(* Logix 5000 project; controller R5_CSS vendor 1 type 14 code 74 rev 19.11; software revision 19.01; part 20 of 20 *)
(* tags used below, declared in another part *)
   FC101 : FLOW_CONTROL;   // QUENCH BASIN FLOW TRANSMITTER CONTROL
   FC101_PIDE : PID_ENHANCED;
   FC140 : FLOW_CONTROL;
   FC140A : FLOW_CONTROL;   // QUENCH TOWER UPPER SPRAY FLOW CONTROL
   FC140B : FLOW_CONTROL;   // QUENCH TOWER LOWER SPRAY FLOW CONTROL
   FC365 : FLOW_CONTROL;   // COALESCER PROCESS IMPURITY FLOW CONTROL
   FT140_TOTAL_FLOW : REAL;
   InputMax_IF8 : REAL;
   InputMin_IF8 : REAL;
   LC101 : LEVEL_CONTROL;   // QUENCH TOWER BASIN LIT
   MyTime : DINT[10];
   P303A : PUMP_CONTROL;
   P303B : PUMP_CONTROL;
   PC132 : PRESSURE_CONTROL;
   PC132_PID : PID;
   PID_FCV365 : PID;
   PID_TCV108_Flow : PID;
   RandomNumber : REAL;
   RandomNumberDint : DINT;
   TC108 : TEMP_CONTROL;   // QUENCH TOWER EXIT GAS TEMPERATURE CONTROL
   TIMER : TIMER[50];   // HX A TIMER FOR START

PROGRAM Simulate   (* main routine MainProgram *)
VAR
   BasinFlowBalance : REAL := 94.5125;
   BasinFlowBalanceAdd : REAL := 0.45176974;
   BasinFlowBalanceAddSCLP : SCLP := (Input := 0.45176974, InputMax := 38.0, ScaledMax := 16000.0, Output := 190.21884);
   BasinFlowBalanceRawAdd : REAL := 190.21884;
   BasinFlowBalanceTmr : TIMER := (PRE := 1000);
   FC140_PID_Sim : AI_Simulate := (ControlVariable := 20.0, AI_Counts := 4025, RandomNumber := 0.637, PID_P := 1.0, PID_I := 1.0, ScaledMin := 4000, ScaledMax := 20000, PID_CV_Min := 20.0, PID_CV_Max := 100.0, UpdateSec := 1.0, DirectActing := 1);
   FC140_SUM : DINT := 4037;
   FC140_SUM_Flow : REAL := 0.46250153;
   FC140_SUM_sclp : SCLP := (Input := 4000.0, InputMin := 4000.0, InputMax := 20000.0, ScaledMax := 200.0);
   FC140A_Flow : REAL := 0.18500061;
   FC140A_SUM : SCLP := (Input := 0.125, InputMax := 200.0, ScaledMin := 4000.0, ScaledMax := 20000.0, Output := 4010.0);
   FC140B_Flow : REAL := 0.27750093;
   FC140B_SUM : SCLP := (Input := 0.25499955, InputMax := 200.0, ScaledMin := 4000.0, ScaledMax := 20000.0, Output := 4020.4);
   FC365_FT_SIM_ENABLE : BOOL;
   FC365_PID_Sim : AI_Simulate := (ControlVariable := 50.0, AI_Counts := 12033, RandomNumber := 0.149, PID_P := 1.0, PID_I := 1.0, ScaledMin := 4000, ScaledMax := 20000, PID_CV_Max := 60.0, UpdateSec := 1.0, DirectActing := 1);
   LC101_PID_Sim : AI_Simulate := (ControlVariable := 2.0, AI_Counts := 4401, RandomNumber := 0.149, PID_P := 1.0, PID_I := 1.0, ScaledMin := 4000, ScaledMax := 20000, PID_CV_Min := 2.0, PID_CV_Max := 100.0, UpdateSec := 1.0, DirectActing := 1);
   PC132_PID_Sim : AI_Simulate := (ControlVariable := 50.0, AI_Counts := 12068, RandomNumber := 0.149, PID_P := 1.0, PID_I := 1.0, ScaledMin := 4000, ScaledMax := 20000, PID_CV_Max := 100.0, UpdateSec := 1.0);
   PC132_SIM_ENABLE : BOOL;
   TEMP_PERCENT : REAL := 50.0;
END_VAR

ROUTINE FC140   (* ladder *)
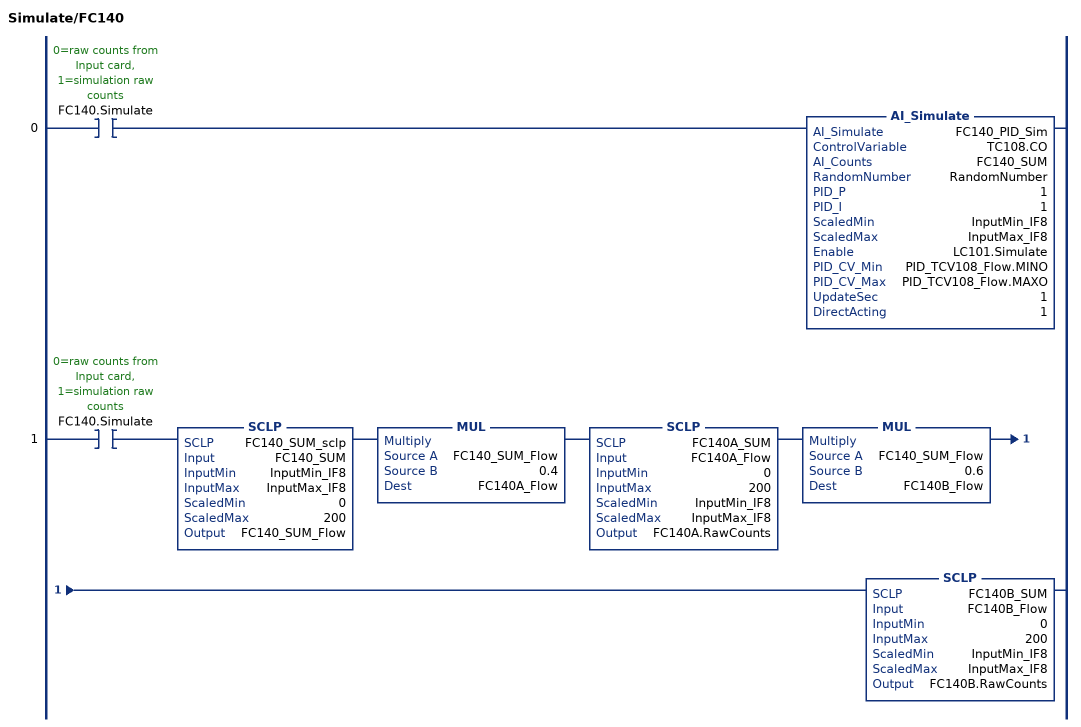
   0: XIC(FC140.Simulate)AI_Simulate(FC140_PID_Sim,TC108.CO,FC140_SUM,RandomNumber,1,1,InputMin_IF8,InputMax_IF8,LC101.Simulate,PID_TCV108_Flow.MINO,PID_TCV108_Flow.MAXO,1,1);
   1: XIC(FC140.Simulate)SCLP(FC140_SUM_sclp,FC140_SUM,InputMin_IF8,InputMax_IF8,0,200,FC140_SUM_Flow)MUL(FC140_SUM_Flow,0.4,FC140A_Flow)SCLP(FC140A_SUM,FC140A_Flow,0,200,InputMin_IF8,InputMax_IF8,FC140A.RawCounts)MUL(FC140_SUM_Flow,0.6,FC140B_Flow)SCLP(FC140B_SUM,FC140B_Flow,0,200,InputMin_IF8,InputMax_IF8,FC140B.RawCounts);
END_ROUTINE

ROUTINE FC365   (* ladder *)
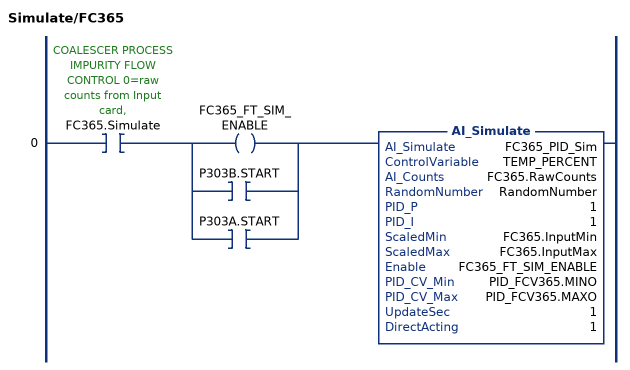
   0: XIC(FC365.Simulate)[OTE(FC365_FT_SIM_ENABLE) ,[XIC(P303B.START) ,XIC(P303A.START) ] ]AI_Simulate(FC365_PID_Sim,TEMP_PERCENT,FC365.RawCounts,RandomNumber,1,1,FC365.InputMin,FC365.InputMax,FC365_FT_SIM_ENABLE,PID_FCV365.MINO,PID_FCV365.MAXO,1,1);
END_ROUTINE

ROUTINE LC101   (* ladder *)
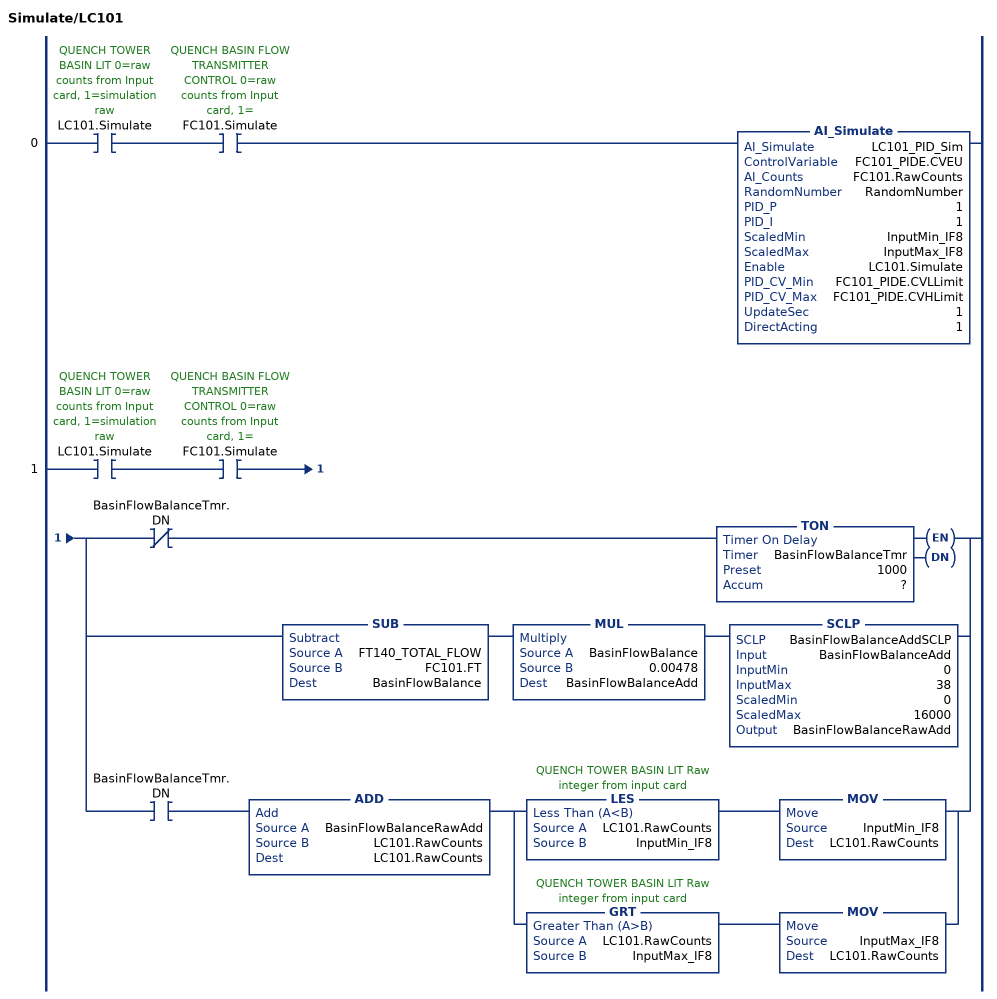
   0: XIC(LC101.Simulate)XIC(FC101.Simulate)AI_Simulate(LC101_PID_Sim,FC101_PIDE.CVEU,FC101.RawCounts,RandomNumber,1,1,InputMin_IF8,InputMax_IF8,LC101.Simulate,FC101_PIDE.CVLLimit,FC101_PIDE.CVHLimit,1,1);
   1: XIC(LC101.Simulate)XIC(FC101.Simulate)[XIO(BasinFlowBalanceTmr.DN) TON(BasinFlowBalanceTmr,?,?) ,SUB(FT140_TOTAL_FLOW,FC101.FT,BasinFlowBalance) MUL(BasinFlowBalance,0.00478,BasinFlowBalanceAdd) SCLP(BasinFlowBalanceAddSCLP,BasinFlowBalanceAdd,0,38,0,16000,BasinFlowBalanceRawAdd) ,XIC(BasinFlowBalanceTmr.DN) ADD(BasinFlowBalanceRawAdd,LC101.RawCounts,LC101.RawCounts) [LES(LC101.RawCounts,InputMin_IF8) MOV(InputMin_IF8,LC101.RawCounts) ,GRT(LC101.RawCounts,InputMax_IF8) MOV(InputMax_IF8,LC101.RawCounts) ] ];
END_ROUTINE

ROUTINE MainProgram   (* ladder *)
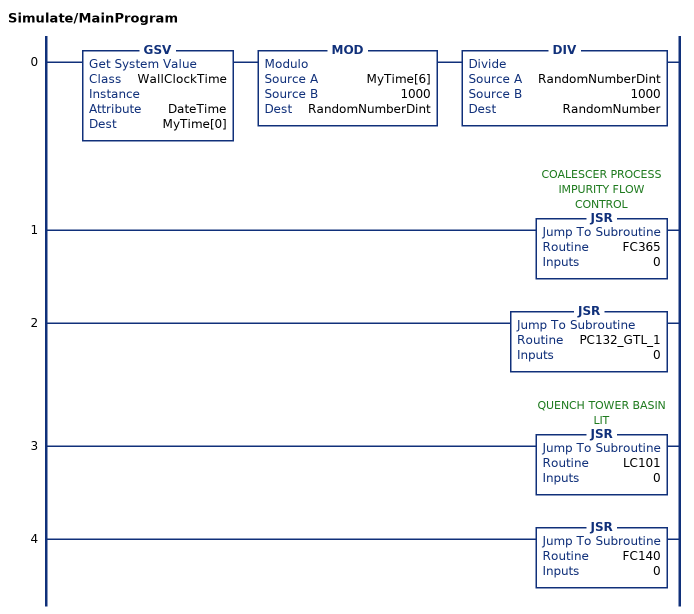
   0: GSV(WallClockTime,,DateTime,MyTime[0])MOD(MyTime[6],1000,RandomNumberDint)DIV(RandomNumberDint,1000,RandomNumber);
   1: JSR(FC365,0);
   2: JSR(PC132_GTL_1,0);
   3: JSR(LC101,0);
   4: JSR(FC140,0);
END_ROUTINE

ROUTINE PC132_GTL_1   (* ladder *)
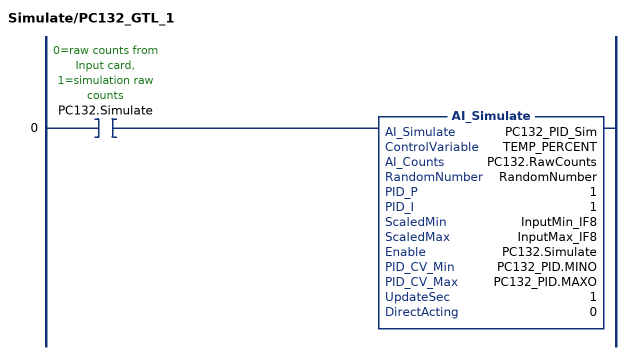
   0: XIC(PC132.Simulate)AI_Simulate(PC132_PID_Sim,TEMP_PERCENT,PC132.RawCounts,RandomNumber,1,1,InputMin_IF8,InputMax_IF8,PC132.Simulate,PC132_PID.MINO,PC132_PID.MAXO,1,0);
END_ROUTINE
END_PROGRAM
